(* PLC project Sin nombre, Desconocido Sin nombre 1 *)
(* stored: creationDateTime 2022-10-17T16:56:25, modificationDateTime 2025-10-23T12:20:35 *)

PROGRAM program0
  VAR
    SENSOR_IR AT %IX0.0 : BOOL := 0;
    SWITCH AT %IX0.1 : BOOL := 0;
    POS_X AT %IW0 : UINT := 500;
    POS_Y AT %IW1 : UINT := 500;
    LED AT %QX0.0 : BOOL := 0;
    RELE AT %QX0.1 : BOOL := 0;
    BOCINA AT %QX0.2 : BOOL := 0;
  END_VAR
  VAR
    SR0 : SR;
    R_TRIG0 : R_TRIG;
    TP0 : TP;
    TOF0 : TOF;
    SR1 : SR;
    R_TRIG1 : R_TRIG;
    ZM_X_LEFT : UINT := 400;
    ZM_X_RIGHT : UINT := 600;
    ZM_Y_TOP : UINT := 600;
    ZM_Y_BOTTOM : UINT := 400;
    TP1 : TP;
    TOF1 : TOF;
  END_VAR

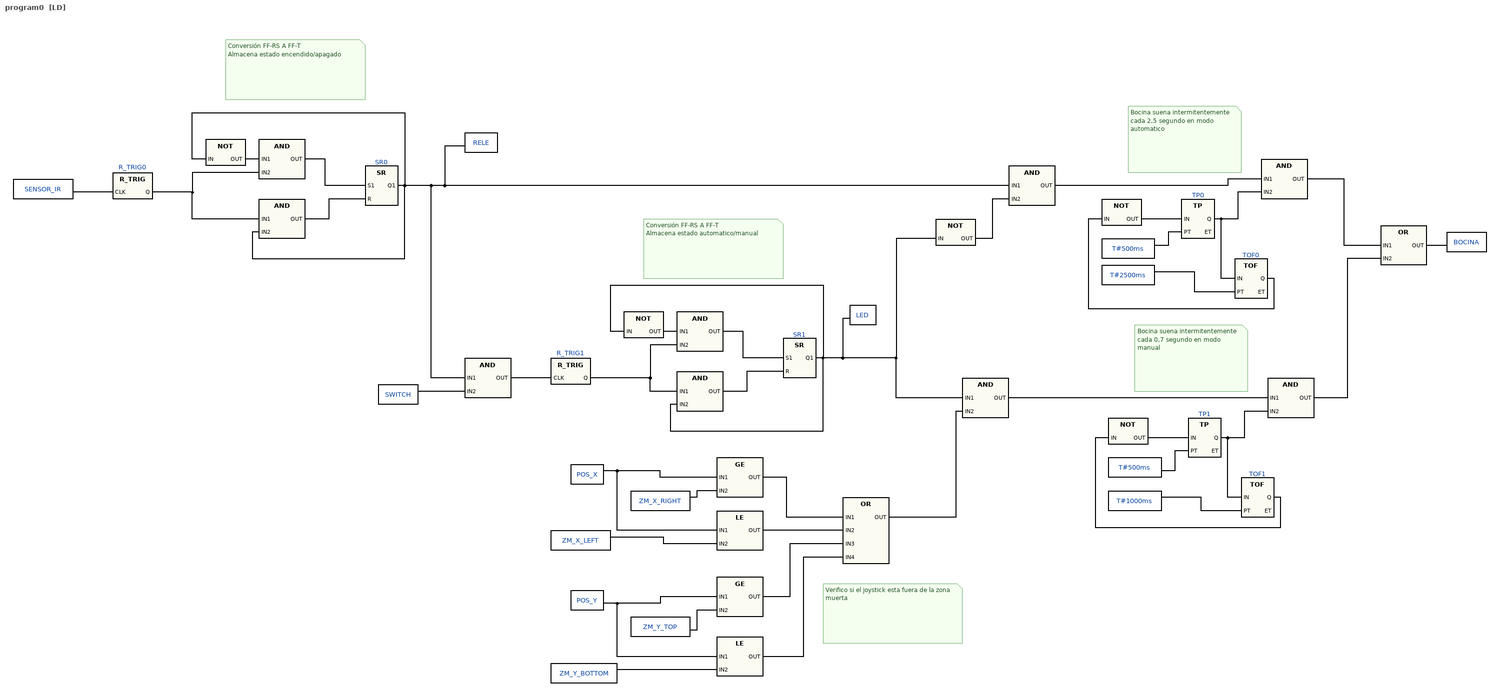
(* LD diagram, written out as Structured Text *)
(* Conversión FF-RS A FF-T
Almacena estado encendido/apagado *)
(* Bocina suena intermitentemente cada 2,5 segundo en modo automatico *)
R_TRIG0(CLK := SENSOR_IR);
SR0(S1 := NOT SR0.Q1 AND R_TRIG0.Q, R := R_TRIG0.Q AND SR0.Q1);
RELE := SR0.Q1;
(* Conversión FF-RS A FF-T
Almacena estado automatico/manual *)
R_TRIG1(CLK := SR0.Q1 AND SWITCH);
SR1(S1 := NOT SR1.Q1 AND R_TRIG1.Q, R := R_TRIG1.Q AND SR1.Q1);
TOF0(IN := TP0.Q, PT := T#2500ms);
TP0(IN := NOT TOF0.Q, PT := T#500ms);
TOF1(IN := TP1.Q, PT := T#1000ms);
TP1(IN := NOT TOF1.Q, PT := T#500ms);
BOCINA := SR0.Q1 AND NOT SR1.Q1 AND TP0.Q OR SR1.Q1 AND (POS_X >= ZM_X_RIGHT OR POS_X <= ZM_X_LEFT OR POS_Y >= ZM_Y_TOP OR POS_Y <= ZM_Y_BOTTOM) AND TP1.Q;
LED := SR1.Q1;
(* Bocina suena intermitentemente cada 0,7 segundo en modo manual *)
(* Verifico si el joystick esta fuera de la zona muerta *)
END_PROGRAM

CONFIGURATION Config0
  RESOURCE Res0 ON PLC
    TASK task0(INTERVAL := T#20ms, PRIORITY := 0);
    PROGRAM instance0 WITH task0 : program0;
  END_RESOURCE
END_CONFIGURATION
